INTERFACE I_ChunkedResponseHeaderAccessor

METHOD PUBLIC TryGetResponseIdFromRequest : BOOL
VAR_INPUT
	Request : I_Request;
	Destination : ANY;
END_VAR
END_METHOD

METHOD PUBLIC TryGetSessionIdFromRequest : BOOL
VAR_INPUT
	Request : I_Request;
	Destination : REFERENCE TO T_MAXSTRING;
END_VAR
END_METHOD

METHOD PUBLIC TryGetSessionIdFromResponse : BOOL
VAR_INPUT
	Response : I_ServerResponse;
	Destination : ANY;
END_VAR
END_METHOD

METHOD PUBLIC UpdateResponseWithHasMoreChunks
VAR_INPUT
	Response : I_ServerResponse;
	ResponseId : T_MAXSTRING;
END_VAR
END_METHOD

END_INTERFACE

(* stored: Version 1.1.0.1, ProductVersion 3.1.4026.13
   Itf I_ChunkedResponseHeaderAccessor: Id {250cb4af-a83e-4d9a-906e-cf45e71db793}
   Method TryGetResponseIdFromRequest: Id {e63ecb7c-930f-487a-931e-37f53e0f4130}
   Method TryGetSessionIdFromRequest: Id {0872ea1c-037f-435a-b101-a9a585396199}
   Method TryGetSessionIdFromResponse: Id {6d2185f9-ad6f-4413-ae6f-b08edda7e87e}
   Method UpdateResponseWithHasMoreChunks: Id {f9c98b2d-bc56-4319-b524-8904d466fcd9} *)
